(* IEC 61131-3 sources: programs/VI-54/VI-54_20171205/VI-54_20171205/Stations/Screen/LseClass170718/Class/FileTransfer_RecvData, 1 file *)

(* ---- FileTransfer_RecvData.st ---- *)
(*!
<Class
	Name               = "FileTransfer_RecvData"
	Revision           = "1.0"
	RealtimeTask       = "false"
	CyclicTask         = "false"
	BackgroundTask     = "false"
	Sigmatek           = "false"
	OSInterface        = "false"
	HighPriority       = "false"
	Automatic          = "false"
	UpdateMode         = "Prescan"
	SharedCommandTable = "true"
	Objectsize         = "(448,120)">
	<Channels>
		<Client Name="cFileTransfer" Required="true" Internal="false"/>
	</Channels>
	<RevDoku>
		<Owner Company="Sigmatek" Author="hötant"/>
		<Dokumentation Revision="1.0" Date="2015-10-15" Author="hötant" Company="Sigmatek" Description="creation of class"/>
	</RevDoku>
	<Network Name="FileTransfer_RecvData">
		<!-- List of Components in this network -->
		<Components>
			<Object
				Name       = "_base"
				Class      = "Comm_RecvData"
				Position   = "(218,120)"
				Visualized = "false">
				<Channels>
					<Server Name="ClassSvr"/>
					<Server Name="sMyID"/>
					<Server Name="sRecvCnt"/>
					<Client Name="cDataMng"/>
				</Channels>
			</Object>
		</Components>
		<Comments>
		</Comments>
		<!-- List of Connections in this network -->
		<Connections>
			<Connection Source="this.ClassSvr" Destination="_base.ClassSvr" Vertices="(1006,210),(834,210),"/>
			<Connection Source="this.sMyID" Destination="_base.sMyID" Vertices="(1006,270),(834,270),"/>
			<Connection Source="this.sRecvCnt" Destination="_base.sRecvCnt" Vertices="(1006,330),(834,330),"/>
			<Connection Source="_base.cDataMng" Destination="this.cDataMng" Vertices="(218,210),(38,210),"/>
		</Connections>
		<!-- Headerfiles -->
		<Options>
		</Options>
	</Network>
</Class>
*)
#pragma using Comm_RecvData

FileTransfer_RecvData : CLASS
: Comm_RecvData
  //Servers:
  //Clients:
	cFileTransfer 	: CltChCmd_FileTransferHandle;
  //Variables:
  //Functions:

	FUNCTION VIRTUAL GLOBAL CallBackReciverCMD
		VAR_INPUT
			DestinationID 	: DINT;
			SourceID 	: DINT;
			size 	: UDINT;
			pdata 	: ^USINT;
			OptCMD 	: USINT;
		END_VAR
		VAR_OUTPUT
			retcode 	: BOOL;
		END_VAR;
  //Tables:
	FUNCTION @STD
		VAR_OUTPUT
			ret_code	: CONFSTATES;
		END_VAR;
	FUNCTION GLOBAL TAB @CT_;
END_CLASS;

#pragma usingLtd FileTransferHandle

FUNCTION VIRTUAL GLOBAL FileTransfer_RecvData::CallBackReciverCMD
	VAR_INPUT
		DestinationID 	: DINT;
		SourceID 	: DINT;
		size 	: UDINT;
		pdata 	: ^USINT;
		OptCMD 	: USINT;
	END_VAR
	VAR_OUTPUT
		retcode 	: BOOL;
	END_VAR

  // Empfangene Daten weiterleiten.
  retcode := cFileTransfer.CallBackReciverCMD(DestinationID, SourceID, size, pdata, OptCMD);

END_FUNCTION
